RoboDK station: ur5_and_table_and_gripper_and_camera.rdk

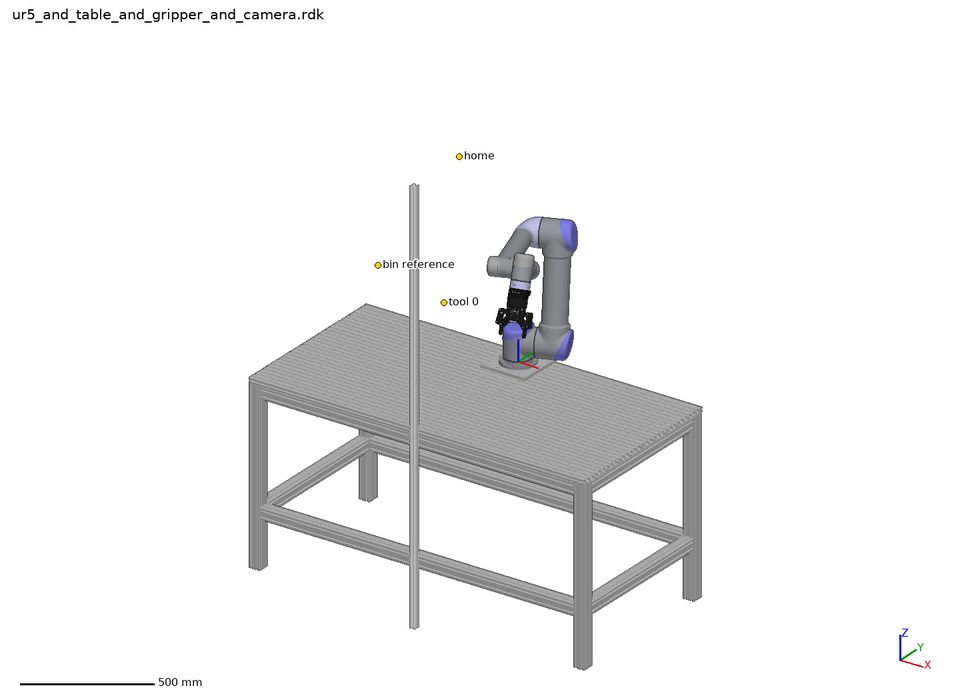
[picture v0: the station drawn from its stored meshes, robots at their saved joint values, targets as dots, program paths as lines]
Station ur5_and_table_and_gripper_and_camera (saved by RoboDK 5.9.0). Poses are relative to the parent item; angles as X-Y-Z fixed-axis rotations.
  - frame UR5 Base at (0, 0, 0) mm
    - robot UR5: 6 axes, payload 5 kg, reach 850 mm, repeatability 0.1 mm, weight 18.4 kg
        modified DH rows (alpha deg, a mm, theta deg, d mm): 0, 0, 0, 89.2; 90, 0, 180, 0; 0, 425, 0, 0; 0, 392.43, 0, 109; -90, 0, 0, 93.65; 90, 0, 180, 82
        joint limits [-360, -360, -360, -360, -360, -360] to [360, 360, 360, 360, 360, 360]; home [0, -90, 90, 0, 90, 0]; saved at [111.869, -100.208, 94.891, 248.63, 266.93, 21.141]
      - tool WRIST_CAMERA_20171116, TCP at (0, 43.75, 11) mm, rotated rx -30 ry 0 rz 0 deg, size 75 x 87.5 x 22.4 mm, geometry from WRIST_CAMERA_20171116.STEP
      - tool GRIPPER_COUPLING, TCP at (0, 0, 190) mm, size 75 x 75 x 16.9 mm
      - tool Gripper RobotiQ 85 Opened, TCP at (0, 0, 190) mm, size 147.4 x 146.8 x 75 mm
    - target home (joint target) at (0, -381, 1000.28) mm, rotated rx -90 ry 0 rz 180 deg; joints [0, -90, 0, -90, 0, 0] of UR5
    - target tool 0 (Cartesian target) at (-75, -375, 375) mm, rotated rx -180 ry 0 rz -180 deg; joints [62.13, -102.576, 81.206, -68.63, -90, -27.87] of UR5
    - target bin reference (Cartesian target) at (-425, -300, 400) mm, rotated rx 180 ry 0 rz -180 deg; joints [23.123, -82.231, 57.897, -65.666, -90, -66.877] of UR5
  - object table_base_setup at (0, 0, 0) mm, rotated rx 0 ry 0 rz -90 deg, size 1524 x 762 x 800.1 mm, geometry from table_base_setup.STEP
  - object 6ft_beam_table at (0, -675, 1000) mm, size 25.4 x 25.4 x 1828.8 mm, geometry from 6ft_beam_table.IGS
